KUKA KRL program: coin2.src, coin2.dat

--- coin2.src ---
&ACCESS RVP
&REL 9
&PARAM DISKPATH = KRC:\R1\3dTisk
&PARAM TEMPLATE = C:\KRC\Roboter\Template\ExpertVorgabe
&PARAM EDITMASK = *
DEF coin2( )

  DECL INT rc
  DECL INT rcNext
  DECL INT pointCount
  DECL BOOL printOk
  DECL BOOL streamOpened
  DECL CHAR fileName[128]
  DECL CNC_MOVE_T point
  DECL CNC_MOVE_T nextPoint


;FOLD PTP HOME Vel=100 % DEFAULT;%{PE}%R 8.2.24,%MKUKATPBASIS,%CMOVE,%VPTP,%P 1:PTP, 2:HOME, 3:, 5:100, 7:DEFAULT
$BWDSTART=FALSE
PDAT_ACT=PDEFAULT
FDAT_ACT=FHOME
BAS(#PTP_PARAMS,100)
$H_POS=XHOME
PTP XHOME
;ENDFOLD

ANOUT ON S_Robot_Vel = 0.1 * $VEL_ACT
s_rq_temp_z_1 = 2300
s_rq_temp_z_2 = 2200
$out[205] = true
$out[206] = false
$out[207] = true


;FOLD LIN P2 Vel=0.5 m/s CPDAT2 Tool[8]:3d tisk tryska Base[8]:3d tisk stul;%{PE}%R 8.2.24,%MKUKATPBASIS,%CMOVE,%VLIN,%P 1:LIN, 2:P2, 3:, 5:0.5, 7:CPDAT2
$BWDSTART=FALSE
LDAT_ACT=LCPDAT2
FDAT_ACT=FP2
BAS(#CP_PARAMS,0.5)
LIN XP2
;ENDFOLD
$VEL.CP = 0.1

;FOLD WAIT Time=0.1 sec;%{PE}%R 8.2.24,%MKUKATPBASIS,%CWAIT,%VWAIT,%P 3:0.1
WAIT SEC 0.1
;ENDFOLD
$out[205] = true

  fileName[] = "coin.txt"
  pointCount = 0
  printOk = TRUE
  streamOpened = FALSE

  ; 1) One-time motion setup for LIN moves.
  rc = Init()
  IF rc == -1 THEN
    MsgNotify("Init failed","prg")
    RETURN
  ENDIF

  ; 2) Open stream from input file.
  rc = CncOpen(fileName[])
  IF rc == -1 THEN
    MsgNotify("CncOpen failed","prg")
    RETURN
  ENDIF
  streamOpened = TRUE

  ; 3) Wait until first point is available, EOF, or error.
  REPEAT
    rc = CncGetNextPoint(point)
    IF rc == 0 THEN
      EXIT
    ENDIF
    IF rc == 1 THEN
      MsgNotify("Empty input file","prg")
      GOTO CLEANUP
    ENDIF
    IF rc == -1 THEN
      MsgNotify("Stream read error","prg")
      printOk = FALSE
      GOTO CLEANUP
    ENDIF
    WAIT SEC 0.01
  UNTIL FALSE

  ; 4) Main processing loop: pipeline next point for approximation.
  REPEAT
    rcNext = CncGetNextPoint(nextPoint)
    IF rcNext == -1 THEN
      MsgNotify("Stream read error","prg")
      printOk = FALSE
      EXIT
    ENDIF

    IF rcNext == 2 THEN
      WAIT SEC 0.01
    ELSE
      IF rcNext == 0 THEN
        rc = MoveLin(point)
        IF rc == -1 THEN
          MsgNotify("MoveLin failed","prg")
          printOk = FALSE
          EXIT
        ENDIF

        pointCount = pointCount + 1
        point = nextPoint
      ELSE
        rc = MoveLinExact(point)
        IF rc == -1 THEN
          MsgNotify("MoveLinExact failed","prg")
          printOk = FALSE
          EXIT
        ENDIF
        pointCount = pointCount + 1
        EXIT
      ENDIF
    ENDIF
  UNTIL FALSE

  IF printOk THEN
    MsgNotify("Print finished, moved points: %1","prg",pointCount)
  ENDIF

CLEANUP:
  ; 5) Cleanup.
  ANOUT OFF S_Robot_Vel
  IF streamOpened THEN
    rc = CncClose()
    IF rc == -1 THEN
      MsgNotify("CncClose failed","prg")
    ENDIF
  ENDIF

END

--- coin2.dat ---
&ACCESS RVP
&REL 9
&PARAM DISKPATH = KRC:\R1\3dTisk
&PARAM TEMPLATE = C:\KRC\Roboter\Template\ExpertVorgabe
&PARAM EDITMASK = *
DEFDAT  coin2
;FOLD EXTERNAL DECLARATIONS;%{PE}%MKUKATPBASIS,%CEXT,%VCOMMON,%P
;FOLD BASISTECH EXT;%{PE}%MKUKATPBASIS,%CEXT,%VEXT,%P
EXT  BAS (BAS_COMMAND  :IN,REAL  :IN )
DECL INT SUCCESS
;ENDFOLD (BASISTECH EXT)
;FOLD USER EXT;%{E}%MKUKATPUSER,%CEXT,%VEXT,%P
;Make your modifications here

;ENDFOLD (USER EXT)
;ENDFOLD (EXTERNAL DECLARATIONS)
DECL BASIS_SUGG_T LAST_BASIS={POINT1[] "P2                      ",POINT2[] "P2                      ",CP_PARAMS[] "CPDAT2                  ",PTP_PARAMS[] "PDAT0                   ",CONT[] "                        ",CP_VEL[] "0.5                     ",PTP_VEL[] "100                     ",SPL_NAME[] "S0                      "}
DECL E6POS XP1={X 358.691589,Y 200.225403,Z -0.0274270307,A 0.0223432798,B -0.00957637932,C -0.0179978702,S 6,T 27,E1 0.0,E2 0.0,E3 0.0,E4 0.0,E5 0.0,E6 0.0}
DECL FDAT FP1={TOOL_NO 8,BASE_NO 8,IPO_FRAME #BASE,POINT2[] " ",TQ_STATE FALSE}
DECL LDAT LCPDAT1={VEL 2.0,ACC 100.0,APO_DIST 100.0,APO_FAC 50.0,AXIS_VEL 100.0,AXIS_ACC 100.0,ORI_TYP #VAR,CIRC_TYP #BASE,JERK_FAC 50.0,GEAR_JERK 50.0,EXAX_IGN 0}
DECL LDAT LCPDAT2={VEL 2.0,ACC 100.0,APO_DIST 100.0,APO_FAC 50.0,AXIS_VEL 100.0,AXIS_ACC 100.0,ORI_TYP #VAR,CIRC_TYP #BASE,JERK_FAC 50.0,GEAR_JERK 50.0,EXAX_IGN 0}
DECL E6POS XP2={X 358.691589,Y 200.225403,Z -0.0274270307,A 0.0223432798,B -0.00957637932,C -0.0179978702,S 6,T 27,E1 0.0,E2 0.0,E3 0.0,E4 0.0,E5 0.0,E6 0.0}
DECL FDAT FP2={TOOL_NO 8,BASE_NO 8,IPO_FRAME #BASE,POINT2[] " ",TQ_STATE FALSE}
ENDDAT
